(* CODESYS project Tc3_Mc3Base.library
   TcLibraryId: Beckhoff Automation GmbH|Tc3_Mc3Base|4.0.17.0
   Company: Beckhoff Automation GmbH
   Title: Tc3_Mc3Base
   Placeholder: Tc3_Mc3Base
   Version: 4.0.17.0

Project tree, tasks and I/O mapping:
  TestCommands/
    function block MC_TriggerError [ST]: FB_init, FB_exit
  Enums/
    data type EBufferMode
    data type ESyncDirection
    data type EReactionToMasterError
    data type EReactionToSlaveError
  Types/
    interface Type_Camming1D: GetCamming1DOid
    interface Type_ErrorTriggerable: GetErrorTriggerableOid
    interface Type_Master1D: GetMaster1DOid
    interface Type_Phasing1D: GetPhasing1DOid
    interface Type_MotionObject: GetMotionObjectOid
  Version/
    global variables Global_Version
*)

// Enums/EBufferMode
(* Buffer mode between buffered commands. *)
{attribute 'TcIecLibraryType'}
{attribute 'Namespace' := 'Tc3_Mc3Base'}
{attribute 'qualified_only'}
{attribute 'strict'}
{attribute 'to_string'}
TYPE EBufferMode : (
	Aborting:=0, 	(* The previous command is aborted and a transition to the new command is initiated immediately. *)
	Buffered:=1	(* The previous command is executed to completion. The new command affects the motion object as 
		soon as the previous movement is 'Done'/'InVelocity'/'InSync'/'InGear'. There is no blending. *)
) UINT;
END_TYPE

// Enums/ESyncDirection
(* Directions in which a slave is allowed to move during synchronizing phase. *)
{attribute 'TcIecLibraryType'}
{attribute 'Namespace' := 'Tc3_Mc3Base'}
{attribute 'qualified_only'}
{attribute 'strict'}
{attribute 'to_string'}
TYPE ESyncDirection : (
		{attribute 'hide'}
Invalid:=0, 	(* Indicates invalid information, e.g. no connection or component not yet ready. *)
	Positive:=1, 	(* Movement is allowed only in positive direction while synchronizing. *)
	Negative:=2, 	(* Movement is allowed only in negative direction while synchronizing. *)
	Both:=3, 	(* Movement is allowed in any direction while synchronizing. *)
	TowardsSlaveSyncPosition:=4	(* Movement is allowed only in direction of the SlaveSyncPosition while synchronizing. *)
) UINT := Invalid;
END_TYPE

// Enums/EReactionToMasterError
(* Reaction type to master errors in master/slave couplings. *)
{attribute 'TcIecLibraryType'}
{attribute 'Namespace' := 'Tc3_Mc3Base'}
{attribute 'qualified_only'}
{attribute 'strict'}
{attribute 'to_string'}
TYPE EReactionToMasterError : (
	TriggerSlaveError:=0, 	(* In case of a master error, a slave error is triggered. *)
	KeepCouplingWithSetValues:=1	(* In case of a master error the coupling is kept with set values and no 
		slave error is triggered. *)
) UINT;
END_TYPE

// Enums/EReactionToSlaveError
(* Reaction type to slave errors in master/slave couplings. *)
{attribute 'TcIecLibraryType'}
{attribute 'Namespace' := 'Tc3_Mc3Base'}
{attribute 'qualified_only'}
{attribute 'strict'}
{attribute 'to_string'}
TYPE EReactionToSlaveError : (
	TriggerMasterError:=0, 	(* In case of a slave error a master error is triggered. *)
	NoReaction:=1	(* No reaction on the master in case of a slave error. *)
) UINT;
END_TYPE

// Version/Global_Version
{attribute 'TcGenerated'}
// This function has been automatically generated from the project information.
VAR_GLOBAL CONSTANT
	{attribute 'const_non_replaced'}
	{attribute 'linkalways'}
	stLibVersion_Tc3_Mc3Base : ST_LibVersion := (iMajor := 4, iMinor := 0, iBuild := 17, iRevision := 0, nFlags := 0, sVersion := '4.0.17.0');
	{attribute 'const_non_replaced'}
	{attribute 'linkalways'}
	sLibraryId_Tc3_Mc3Base : String := 'Beckhoff Automation GmbH|Tc3_Mc3Base|4.0.17.0';
END_VAR

// TestCommands/MC_TriggerError

{attribute 'c++_compatible'}
{attribute 'external_name' := 'MC_TriggerError_GUID_64D28803_CE42_C2F4_631F_C5998BDC03BE'}
{attribute 'TcIecLibraryType'}
{attribute 'hide_all_locals'}
(* 
		This function block triggers an error in the target motion object.
	 *)
FUNCTION_BLOCK MC_TriggerError
VAR_INPUT
	(* Interface pointer to the object on which the error should be triggered (e.g. Axis). *)
	{attribute 'GUID' := 'A3E57B21-F9C4-4D38-B5E2-1F4E8A2B6C9D'}
	{attribute 'Namespace' := 'Tc3_Mc3Base'}
	MotionObject : Type_ErrorTriggerable;
	(* Trigger the command with rising edge. *)
	Execute : BOOL;
END_VAR
VAR
	 {attribute 'hide'}
	_reserved1 : ARRAY [1..3] OF USINT;
END_VAR
VAR_INPUT
	(* Error code to be triggered *)
	ErrorCode : UDINT;
	(* Trigger a ControlError (MC has no control over the axis, i.e. hardware or communication fault). *)
	ControlError : BOOL;
END_VAR
VAR_OUTPUT
	(* Error has been successfully triggered. *)
	Done : BOOL;
	(* Function block is not finished and new output values are to be expected. *)
	Busy : BOOL;
	(* Error occurred within function block. *)
	Error : BOOL;
	(* Error identifier *)
	ErrorId : UDINT;
END_VAR
VAR
	 {attribute 'hide'}
	_reserved2 : UINT_0_32;
	 {attribute 'hide'}
	_reserved3 : ARRAY [1..36] OF UINT_8_16;
	 {attribute 'hide'}
	_reserved4 : ARRAY [1..12] OF USINT;
END_VAR

{attribute 'TcTypeSystem'}

(* Internal method *)
{attribute 'hide'}
METHOD FB_init : BOOL
VAR_INPUT
	(*  if TRUE, the retain variables are initialized (warm start / cold start) *)
	bInitRetains : BOOL;
	(*  if TRUE, the instance afterwards gets moved into the copy code (online change) *)
	bInCopyCode : BOOL;
END_VAR
END_METHOD

{attribute 'TcTypeSystem'}

(* Internal method *)
{attribute 'hide'}
METHOD FB_exit : BOOL
VAR_INPUT
	(*  if TRUE, the exit method is called for exiting an instance that is copied afterwards (online change). *)
	bInCopyCode : BOOL;
END_VAR
END_METHOD

END_FUNCTION_BLOCK

// Types/Type_ErrorTriggerable
(* Type for a motion control object that supports error triggering (e. g. supported by AXIS_REF). *)
{attribute 'Namespace' := 'Tc3_Mc3Base'}
{attribute 'hide'}
{attribute 'c++_compatible'}
INTERFACE Type_ErrorTriggerable

{attribute 'TcTypeSystem'}
{attribute 'c++_compatible'}
{attribute 'minimal_input_size' := '4'}
{attribute 'pack_mode' := '4'}
{attribute 'hide'}
METHOD GetErrorTriggerableOid : GLOBAL.OTCID
END_METHOD

END_INTERFACE

// Types/Type_Camming1D
(* Type for a motion control object that can operate as a 1D camming slave object (like slave axis for MC_CamIn, e. g. supported by AXIS_REF). *)
{attribute 'Namespace' := 'Tc3_Mc3Base'}
{attribute 'c++_compatible'}
INTERFACE Type_Camming1D

{attribute 'TcTypeSystem'}
{attribute 'c++_compatible'}
{attribute 'minimal_input_size' := '4'}
{attribute 'pack_mode' := '4'}
{attribute 'hide'}
METHOD GetCamming1DOid : GLOBAL.OTCID
END_METHOD

END_INTERFACE

// Types/Type_Master1D
(* Type for a motion control object that can operate as a 1D master object (like master axis for MC_GearIn, e. g. supportet by AXIS_REF). *)
{attribute 'Namespace' := 'Tc3_Mc3Base'}
{attribute 'c++_compatible'}
INTERFACE Type_Master1D

{attribute 'TcTypeSystem'}
{attribute 'c++_compatible'}
{attribute 'minimal_input_size' := '4'}
{attribute 'pack_mode' := '4'}
{attribute 'hide'}
METHOD GetMaster1DOid : GLOBAL.OTCID
END_METHOD

END_INTERFACE

// Types/Type_Phasing1D
(* Type for a motion control object that supports 1D phasing (MC_PhasingAbsolute, e. g. supported by AXIS_REF). *)
{attribute 'Namespace' := 'Tc3_Mc3Base'}
{attribute 'c++_compatible'}
INTERFACE Type_Phasing1D

{attribute 'TcTypeSystem'}
{attribute 'c++_compatible'}
{attribute 'minimal_input_size' := '4'}
{attribute 'pack_mode' := '4'}
{attribute 'hide'}
METHOD GetPhasing1DOid : GLOBAL.OTCID
END_METHOD

END_INTERFACE

// Types/Type_MotionObject
{attribute 'Namespace' := 'Tc3_Mc3Base'}
{attribute 'c++_compatible'}
INTERFACE Type_MotionObject

{attribute 'TcTypeSystem'}
{attribute 'c++_compatible'}
{attribute 'minimal_input_size' := '4'}
{attribute 'pack_mode' := '4'}
{attribute 'hide'}
METHOD GetMotionObjectOid : GLOBAL.OTCID
END_METHOD

END_INTERFACE
